% RSLogix 500 project Aquatic Outside Pool - 16-10-08.RSS, saved by version 7.00.00.19 %
PROJECT "AQUATIC2"    % processor: Bul.1763 MicroLogix 1100 Series A %

PROGRAM FILES
  LAD 2 "MAIN"  5 rungs
  LAD 3 "SCALING"  4 rungs
  LAD 4 "PID"  5 rungs

DATA FILES
  O0 OUTPUT  6 elements
  I1 INPUT  12 elements
  S2 STATUS  66 elements
  B3 BINARY  1 elements
  T4 TIMER  1 elements
  C5 COUNTER  1 elements
  R6 CONTROL  1 elements
  N7 INTEGER  24 elements
  F8 FLOAT  1 elements
  PD9   1 elements

LADDER 2 "MAIN"
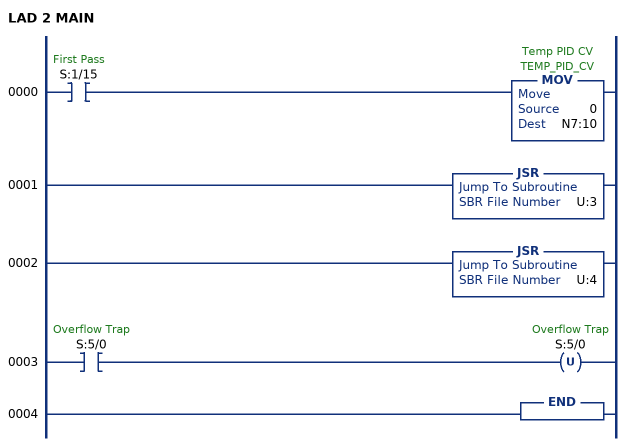
% Rung: 0 %
SOR XIC S:1/15 MOV 0 N7:10 EOR
%   S:1/15  "First Pass" %
%   N7:10  TEMP_PID_CV  "Temp PID CV" %
% Rung: 1 %
SOR JSR U:3 EOR
% Rung: 2 %
SOR JSR U:4 EOR
% Rung: 3 %
SOR XIC S:5/0 OTU S:5/0 EOR
%   S:5/0  "Overflow Trap" %
% Rung: 4 %
SOR END EOR

LADDER 3 "SCALING"
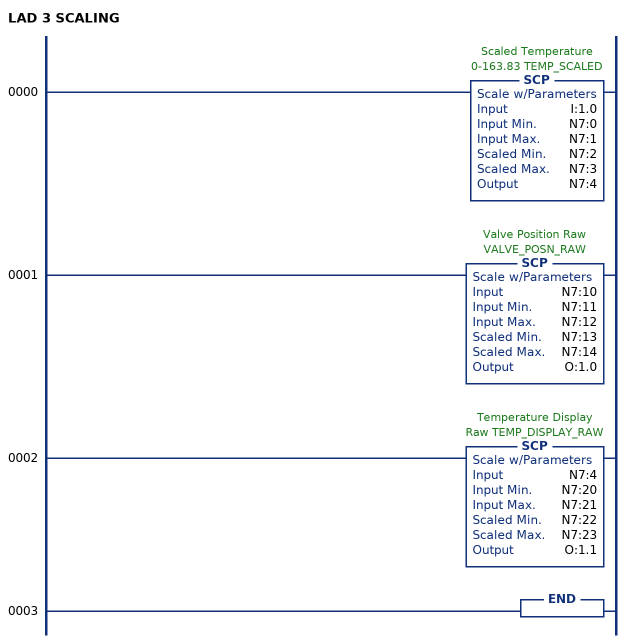
% Rung: 0 %
SOR SCP I:1.0 N7:0 N7:1 N7:2 N7:3 N7:4 EOR
%   I:1.0  TEMP  "Temperature Analog Raw" %
%   N7:4  TEMP_SCALED  "Scaled Temperature 0-163.83" %
% Rung: 1 %
SOR SCP N7:10 N7:11 N7:12 N7:13 N7:14 O:1.0 EOR
%   N7:10  TEMP_PID_CV  "Temp PID CV" %
%   O:1.0  VALVE_POSN_RAW  "Valve Position Raw" %
% Rung: 2 %
SOR SCP N7:4 N7:20 N7:21 N7:22 N7:23 O:1.1 EOR
%   N7:4  TEMP_SCALED  "Scaled Temperature 0-163.83" %
%   O:1.1  TEMP_DISPLAY_RAW  "Temperature Display Raw" %
% Rung: 3 %
SOR END EOR

LADDER 4 "PID"
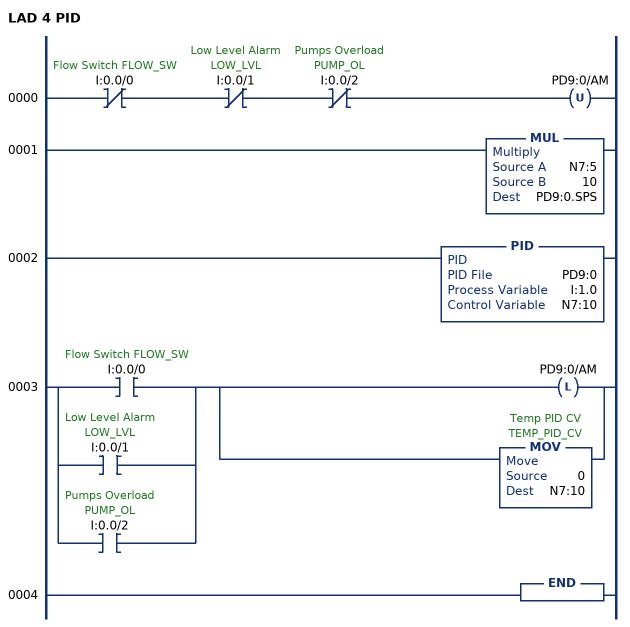
% Rung: 0 %
SOR XIO I:0.0/0 XIO I:0.0/1 XIO I:0.0/2 OTU PD9:0/AM EOR
%   I:0.0/0  FLOW_SW  "Flow Switch" %
%   I:0.0/1  LOW_LVL  "Low Level Alarm" %
%   I:0.0/2  PUMP_OL  "Pumps Overload" %
% Rung: 1 %
SOR MUL N7:5 10 PD9:0.SPS EOR
% Rung: 2 %
SOR PID PD9:0 I:1.0 N7:10 EOR
%   I:1.0  TEMP  "Temperature Analog Raw" %
%   N7:10  TEMP_PID_CV  "Temp PID CV" %
% Rung: 3 %
SOR BST XIC I:0.0/0 NXB XIC I:0.0/1 NXB XIC I:0.0/2 BND BST OTL PD9:0/AM NXB MOV 0 N7:10 BND EOR
%   I:0.0/0  FLOW_SW  "Flow Switch" %
%   I:0.0/1  LOW_LVL  "Low Level Alarm" %
%   I:0.0/2  PUMP_OL  "Pumps Overload" %
%   N7:10  TEMP_PID_CV  "Temp PID CV" %
% Rung: 4 %
SOR END EOR

DATA TABLE (non-zero values as saved)
DATA N7
% N7:0 % 0 16383 0 5000 3081 275 1250 0 0 0
% N7:10 % 0 0 16383 3276 16383 0 0 0 0 0
% N7:20 % 0 5000 3276 16383
